{attribute 'GeneratedUsingTerminal: EL5122-0000-0016'}
{attribute addProperty BoxType "EL5122-0000-0016"}
{attribute addProperty Id "ControlAT %Q*Control_A35B59FC6Set_counter_valueAT %Q*UDINT4"}
{attribute addProperty CRC "3106965037"}
{attribute addProperty Size "10"}
TYPE ENC_Control_Channel_B930862D :
STRUCT
	{attribute addProperty Name "Control"}
	Control AT %Q* : Control_A35B59FC;
	{attribute addProperty Name "Set_counter_value"}
	Set_counter_value AT %Q* : UDINT;
END_STRUCT
END_TYPE

(* stored: Version 1.2.0.0, ProductVersion 3.1.4024.9
   DUT ENC_Control_Channel_B930862D: Id {0cd244d5-9449-47ee-91f9-958cebc55215} *)
